// TIA Portal project "Push button for conveyor motor" (V20)

(* hardware
DEVICE "S7-1500/ET200MP station_1"  S7-1500 station
   slot 0: "Rail_0"  Rack  6ES7 590-1***0-0AA0
   slot 1: "PLC_1"  CPU 1512C-1 PN  6ES7 512-1CK00-0AB0  V2.9
      slot 3: "CPU display_1"  6ES7591-1AA00-0AA0
      slot 32768: "PROFINET interface_1"  X1
         slot 32769: "Port_1"  X1 P1
         slot 32770: "Port_2"  X1 P2
      slot 34817: "Virtual CP interface port_1"  Virtual CP interface port  Virtual CP interface port
*)

// ===== PLC "PLC_1"  CPU 1512C-1 PN =====

VAR_GLOBAL   // PLC tag table "Default tag table"
   "Push Button" AT %I10.0 : Bool;
   "Conveyor Motor" AT %Q4.0 : Bool;
   "Memory 1" AT %Q4.1 : Bool;
   "Memory 2" AT %Q4.2 : Bool;
   "Memory 3" AT %Q4.3 : Bool;
END_VAR

ORGANIZATION_BLOCK "Main"   // OB1, LAD, ProgramCycle
TITLE = "Main Program Sweep (Cycle)"
{ S7_Optimized_Access := 'TRUE' }
VERSION : 0.1
   VAR_INPUT
      Initial_Call : Bool;   // Initial call of this OB
      Remanence : Bool;   // =True, if remanent data are available
   END_VAR
BEGIN

REGION Network 1: Push Button for conveyor motor
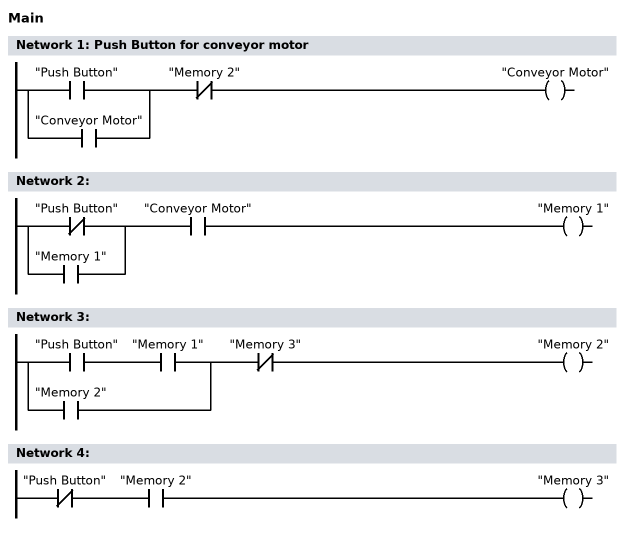
   RUNG wire#powerrail
      Contact( "Push Button" )
      wire#w1
      I_Contact( "Memory 2" )
      Coil( "Conveyor Motor" )
   END_RUNG
   RUNG wire#powerrail
      Contact( "Conveyor Motor" )
   END_RUNG wire#w1
   // the same network as SCL:
   "Conveyor Motor" := ("Push Button" OR "Conveyor Motor") AND NOT "Memory 2";
END_REGION

REGION Network 2
   RUNG wire#powerrail
      I_Contact( "Push Button" )
      wire#w1
      Contact( "Conveyor Motor" )
      Coil( "Memory 1" )
   END_RUNG
   RUNG wire#powerrail
      Contact( "Memory 1" )
   END_RUNG wire#w1
   // the same network as SCL:
   "Memory 1" := (NOT "Push Button" OR "Memory 1") AND "Conveyor Motor";
END_REGION

REGION Network 3
   RUNG wire#powerrail
      Contact( "Push Button" )
      Contact( "Memory 1" )
      wire#w1
      I_Contact( "Memory 3" )
      Coil( "Memory 2" )
   END_RUNG
   RUNG wire#powerrail
      Contact( "Memory 2" )
   END_RUNG wire#w1
   // the same network as SCL:
   "Memory 2" := (("Push Button" AND "Memory 1") OR "Memory 2") AND NOT "Memory 3";
END_REGION

REGION Network 4
   RUNG wire#powerrail
      I_Contact( "Push Button" )
      Contact( "Memory 2" )
      Coil( "Memory 3" )
   END_RUNG
   // the same network as SCL:
   "Memory 3" := NOT "Push Button" AND "Memory 2";
END_REGION
END_ORGANIZATION_BLOCK